(*
    This FB tests the free function TEST_FINISHED_NAMED. Calling this function with a name that doesn't exist should
    produce an error message that says so. This error message should also only be printed once.
*)
{attribute 'call_after_init'}
FUNCTION_BLOCK FB_TestFinishedNamedDoesNotExist EXTENDS TcUnit.FB_TestSuite
VAR
END_VAR

Test_FinishedNamed();

METHOD PRIVATE Test_FinishedNamed
VAR
    a : INT := 2;
    b : INT := 2;
    
    bajs : BOOL;
END_VAR
TEST('Test_FinishedNamed');

AssertEquals_INT(Expected := a,
                 Actual := b,
                 Message := 'Values differ');

TEST_FINISHED_NAMED('AnotherTestNameThatDoesNotExist');
END_METHOD

END_FUNCTION_BLOCK

(* stored: Version 1.1.0.1, ProductVersion 3.1.4022.18
   POU FB_TestFinishedNamedDoesNotExist: Id {35a9595b-53ed-4b98-952e-2505a213e9de}, SpecialFunc None
   Method Test_FinishedNamed: Id {cfb93715-88e1-42c4-9031-f3f7c5b1a64a} *)
